// TIA Portal V19 export
DATA_BLOCK "A0302_PareggiatoreCoda"   // DB152
// stored: InstanceOfName A0302_PareggiatoreCoda_FB, InstanceOfType FB
"A0302_PareggiatoreCoda_FB"
   // VAR_INPUT
   //    AreaInterface : "AreaInterface";
   //    ZSI : "udt_ZoneSafetyInterface";
   //    DSI_Feed : "udt_DeviceSafetyInterface";
   //    DSI_Valve : "udt_DeviceSafetyInterface";
   //    DSI_OilValve : "udt_DeviceSafetyInterface";
   //    Drive : "TAx_DriveInterface";
   //    DataIn : Struct
   //       OP_MoveToPos : Bool;
   //       BattutaVrt : Struct
   //          OP : "OP_PB";
   //       END_STRUCT;
   //       PareggLong : Struct
   //          OP : "OP_PB";
   //          AnalSens : Int;
   //       END_STRUCT;
   //       Sens { ExternalWritable := 'False'} : Struct
   //          FTC_Ingombro_In : Bool;
   //          FTC_Ingombro_Out : Bool;
   //          PresenzaMat : Bool;
   //          FC_Aticoll_Spalla : Bool;
   //       END_STRUCT;
   //    END_STRUCT;
   //    CIn : Struct
   //       Manager : Struct
   //          EnableStopDoorOpeningReq { ExternalAccessible := 'False'; ExternalVisible := 'False'; ExternalWritable := 'False'} : Bool;
   //          EnableStopInPhase { ExternalAccessible := 'False'; ExternalVisible := 'False'; ExternalWritable := 'False'} : Bool;
   //          EnableStopProgrammed { ExternalAccessible := 'False'; ExternalVisible := 'False'; ExternalWritable := 'False'} : Bool;
   //          Control_ON { ExternalAccessible := 'False'; ExternalVisible := 'False'; ExternalWritable := 'False'} : Bool;
   //          MoveToPos { ExternalAccessible := 'False'; ExternalVisible := 'False'; ExternalWritable := 'False'} : Bool;
   //          Pos { ExternalAccessible := 'False'; ExternalVisible := 'False'; ExternalWritable := 'False'} : LReal;
   //          Speed : LReal;
   //          Bloccaggio { ExternalAccessible := 'False'; ExternalVisible := 'False'; ExternalWritable := 'False'} : Struct
   //             Rest : Bool;
   //             Work : Bool;
   //          END_STRUCT;
   //          BattutaVrt { ExternalAccessible := 'False'; ExternalVisible := 'False'; ExternalWritable := 'False'} : Struct
   //             Rest : Bool;
   //             Work : Bool;
   //          END_STRUCT;
   //          PareggLong { ExternalAccessible := 'False'; ExternalVisible := 'False'; ExternalWritable := 'False'} : Struct
   //             Rest : Bool;
   //             Work : Bool;
   //          END_STRUCT;
   //       END_STRUCT;
   //       SemiAut_Pb { ExternalWritable := 'False'} : Bool;
   //       Bordatrice : Struct
   //          Ax : "Positioning_EPOS_Machine_COut";
   //          Sts : Struct
   //             PosTargetEnable : Bool;
   //             PosTarget_Reached : Bool;
   //             In_W_Pos : Bool;
   //             AtRest : Bool;
   //          END_STRUCT;
   //          RegSpalla : Struct
   //             Infeed_ReqON : Bool;
   //          END_STRUCT;
   //       END_STRUCT;
   //       Rulliera { ExternalWritable := 'False'} : Struct
   //          Ax_1 : "SpeedMachine_COut";
   //          Ax_2 : "SpeedMachine_COut";
   //          Centratori : "ValveMachine_COut";
   //          Coda : Struct
   //             Sens : Struct
   //                FTC_Rall : Bool;
   //                FTC_Prox_Ing : Bool;
   //             END_STRUCT;
   //          END_STRUCT;
   //          Centro : Struct
   //             Sens : Struct
   //                FTC_Centrale : Bool;
   //             END_STRUCT;
   //          END_STRUCT;
   //       END_STRUCT;
   //       CarroPareggCoda : Struct
   //          Pareggia : Bool;
   //          OilInTargetPressure { ExternalWritable := 'False'} : Bool;
   //       END_STRUCT;
   //       CarroPareggTesta { ExternalWritable := 'False'} : Struct
   //          Sens : Struct
   //             FTC1_Rall : Bool;
   //             FTC2_Prox_Ls : Bool;
   //             PresenzaMat : Bool;
   //          END_STRUCT;
   //       END_STRUCT;
   //       CarriPareggiatori : Struct
   //          ZoneA0302Entry_Empty { ExternalWritable := 'False'} : Bool;
   //          ZoneA0302Exit_Empty { ExternalWritable := 'False'} : Bool;
   //          RequestNewPosition : Bool;
   //       END_STRUCT;
   //       Spalle : Struct
   //          Coda : Struct
   //             ActualPos : LReal;
   //          END_STRUCT;
   //          Testa : Struct
   //             ActualPos : LReal;
   //          END_STRUCT;
   //       END_STRUCT;
   //       Manipolatore : Struct
   //          Sollevatore : "ValveMachine_COut";
   //       END_STRUCT;
   //       Centratori : Struct
   //          Sollevamento : "ValveMachine_COut";
   //       END_STRUCT;
   //    END_STRUCT;
   //    Config : Struct
   //       Ax : "Positioning_DOL_Machine_Config";
   //       Bloccaggio : "ValveMachine_Config";
   //       BattutaVerticale : "ValveMachine_Config";
   //       PareggiatoreLong : "ValveMachine_Config";
   //       PosPareggiatore : Struct
   //          QuotaMin_Work : LReal;
   //          QuotaMax_Work : LReal;
   //       END_STRUCT;
   //       MinDistanzaConSpalla : LReal;
   //       DelayMissingCondition : Time;
   //    END_STRUCT;
   //    HWID : Struct
   //       Ax_TEL1 : HW_SUBMODULE;
   //       Enc_IO : HW_SUBMODULE;
   //    END_STRUCT;
   // END_VAR
   // VAR_OUTPUT
   //    MachineInterface : "MachineInterface";
   //    COut : Struct
   //       Ax : "Positioning_DOL_Machine_COut";
   //       Bloccaggio : "ValveMachine_COut";
   //       BattutaVerticale : "ValveMachine_COut";
   //       PareggiatoreLong : "ValveMachine_COut";
   //       Ax_InWPos : Bool;
   //       Anticipi : Struct
   //          Work : Struct
   //             BattutaVrt : Bool;
   //             PareggLong : Bool;
   //          END_STRUCT;
   //          Rest : Struct
   //             BattutaVrt : Bool;
   //             PareggLong : Bool;
   //          END_STRUCT;
   //       END_STRUCT;
   //    END_STRUCT;
   // END_VAR
   // VAR_IN_OUT
   //    Par : Struct
   //       Ax : "Positioning_DOL_Machine_Par";
   //       Ax_Pers : "Positioning_DOL_Machine_Pers_Data";
   //       Enc : "PosFbk_RTN";
   //       Ax_Aut : "A0301_Mach_Speed_Par";
   //       Bloccaggio_Sens : Struct
   //          "2191B1" : "Analogic_SensorManagement_Par";
   //          SogliaWork : Real;
   //       END_STRUCT;
   //       CarroPareggCoda : Struct
   //          Delay_StartMove : Time;
   //          Preset : LReal;
   //       END_STRUCT;
   //       Cremaliera : Struct
   //          Modulo : LReal;
   //          Passo : LReal;
   //       END_STRUCT;
   //    END_STRUCT;
   //    Par_Sens : Struct
   //       AI : "Analogic_SensorManagement_Par";
   //    END_STRUCT;
   //    Data_Sens : "Analogic_SensorManagement_Data";
   //    Par_MachSens : "A0301_Mach_Sens_Par";
   //    IEC_SP : Struct
   //       FTC_Input : Struct
   //          TON_PT : Time;
   //          TOF_PT : Time;
   //       END_STRUCT;
   //       FTC_Output : Struct
   //          TON_PT : Time;
   //          TOF_PT : Time;
   //       END_STRUCT;
   //       FTC_PresentMat : Struct
   //          TON_PT : Time;
   //          TOF_PT : Time;
   //       END_STRUCT;
   //       Check_2119B1 : Struct
   //          TON_PT : Time;
   //       END_STRUCT;
   //    END_STRUCT;
   // END_VAR
   // VAR
   //    Alarm : Struct
   //       Ax : "Positioning_DOL_Machine_Alr";
   //       Enc : "PosFbk_Encoder_Alr";
   //       Bloccaggio : "ValveAlr";
   //       BattutaVerticale : "ValveAlr";
   //       PareggiatoreLong : "ValveAlr";
   //       PareggLong_AnalSens_Issue : Bool;
   //       SensFC_Aticoll_Spalla : Bool;
   //       Bloccaggio_AnalSens_Issue : Bool;
   //    END_STRUCT;
   //    Warning : Struct
   //       Ax : "Positioning_DOL_Machine_Wng";
   //       Bloccaggio : "ValveMachine_Wng";
   //       BattutaVerticale : "ValveMachine_Wng";
   //       PareggiatoreLongitudinale : "ValveMachine_Wng";
   //       PosPareggiatoreLong : "Analogic_SensorManagement_Warning";
   //       MissingCnd : Struct
   //          OP_REST_BattutaVrt : Bool;
   //          OP_WORK_BattutaVrt : Bool;
   //          OP_REST_PareggLong : Bool;
   //          OP_WORK_PareggLong : Bool;
   //          OP_REST_Bloccaggio : Bool;
   //          OP_WORK_Bloccaggio : Bool;
   //       END_STRUCT;
   //       SW_Limit_AntiCollision : Bool;
   //    END_STRUCT;
   //    HMI : Struct
   //       AnalogSensor : "AnalogSens_HmiData";
   //       Ax : Struct
   //          PbPreset : Bool;
   //          B_Preset_UM2 : Bool;
   //          PresetValue : LReal;
   //       END_STRUCT;
   //    END_STRUCT;
   //    Sts : Struct
   //       ReadyForMove : Bool;
   //       OP_PCoda_CanMoveFreely : Bool;
   //       OP_Ax_CanMoveFreely : Bool;
   //       Op_MoveToPos_Cnd : Bool;
   //       BattutaVrt : Struct
   //          OP_Rest_Cnd : Bool;
   //          Op_Work_Cnd : Bool;
   //       END_STRUCT;
   //       PareggLong : Struct
   //          OP_Rest_Cnd : Bool;
   //          Op_Work_Cnd : Bool;
   //       END_STRUCT;
   //    END_STRUCT;
   //    Ctrl : Struct
   //       BattutaVrt : Struct
   //          OP_Rest_Man : Bool;
   //          OP_Work_Man : Bool;
   //          OP_Rest_Aut : Bool;
   //          OP_Work_Aut : Bool;
   //          OP_Rest : Bool;
   //          OP_Work : Bool;
   //       END_STRUCT;
   //       PareggLong : Struct
   //          CheckMesure : Bool;
   //          OP_Rest_Aut : Bool;
   //          OP_Work_Aut : Bool;
   //          OP_Rest_Man : Bool;
   //          OP_Work_Man : Bool;
   //          OP_Rest : Bool;
   //          OP_Work : Bool;
   //       END_STRUCT;
   //       Ax : Struct
   //          OP_MoveToPos_Man : Bool;
   //          OP_MoveToPos_Aut : Bool;
   //          OP_MoveToPos : Bool;
   //       END_STRUCT;
   //    END_STRUCT;
   //    AUX : Struct
   //       OP_MoveToPos : Bool;
   //       BattutaVrt : Struct
   //          OP_Rest : Bool;
   //          OP_Work : Bool;
   //       END_STRUCT;
   //       PareggLong : Struct
   //          OP_Rest : Bool;
   //          OP_Work : Bool;
   //       END_STRUCT;
   //    END_STRUCT;
   //    Ax { S7_SetPoint := 'True'} : "Positioning_DOL_Machine_FB";
   //    Enc : "PosFbk_SickAFM60";
   //    Enc_ITF : "PosFbk_ITF";
   //    Bloccaggio { S7_SetPoint := 'True'} : "ValveMachine_FB";
   //    BattutaVerticale { S7_SetPoint := 'True'} : "ValveMachine_FB";
   //    PareggiatoreLong { S7_SetPoint := 'True'} : "ValveMachine_FB";
   //    PosPareggLong { S7_SetPoint := 'True'} : "Analogic_SensorManagement";
   //    TON_PareggLong : Struct
   //       OP_REST_MissingCnd { S7_SetPoint := 'True'} : TON_TIME;
   //       OP_WORK_MissingCnd { S7_SetPoint := 'True'} : TON_TIME;
   //    END_STRUCT;
   //    TON_BattutaVrt : Struct
   //       OP_REST_MissingCnd { S7_SetPoint := 'True'} : TON_TIME;
   //       OP_WORK_MissingCnd { S7_SetPoint := 'True'} : TON_TIME;
   //    END_STRUCT;
   //    TON_Bloccaggio : Struct
   //       OP_REST_MissingCnd { S7_SetPoint := 'True'} : TON_TIME;
   //       OP_WORK_MissingCnd { S7_SetPoint := 'True'} : TON_TIME;
   //    END_STRUCT;
   //    IEC_FTC_Input : Struct
   //       TON_Delay : IEC_TIMER;
   //       TOF_Delay { S7_SetPoint := 'True'} : IEC_TIMER;
   //       FTC_On { S7_SetPoint := 'True'} : Bool;
   //    END_STRUCT;
   //    IEC_FTC_Output : Struct
   //       TON_Delay : IEC_TIMER;
   //       TOF_Delay { S7_SetPoint := 'True'} : IEC_TIMER;
   //       FTC_On { S7_SetPoint := 'True'} : Bool;
   //    END_STRUCT;
   //    IEC_FTC_PresentMat : Struct
   //       TON_Delay : IEC_TIMER;
   //       TOF_Delay { S7_SetPoint := 'True'} : IEC_TIMER;
   //       FTC_On { S7_SetPoint := 'True'} : Bool;
   //    END_STRUCT;
   //    IEC_DelayCheck_2119B1 : IEC_TIMER;
   //    Bloccaggio_AnalSens { S7_SetPoint := 'True'} : "AnalogThreshold";
   //    CarroCoda { ExternalAccessible := 'False'; ExternalVisible := 'False'; ExternalWritable := 'False'} : Struct
   //       RimanenzaPos : LReal;
   //       PassoReq : LReal;
   //       PosBattutePz : LReal;
   //       SemiBeamLen : LReal;
   //       NrPassiReq : LReal;
   //       Pos : LReal;
   //    END_STRUCT;
   //    TON_DistanzaOK : IEC_TIMER;
   //    TON_Anticipi : Struct
   //       Rest : Struct
   //          BattutaVrt { S7_SetPoint := 'True'} : IEC_TIMER;
   //          PareggLong : IEC_TIMER;
   //       END_STRUCT;
   //       Work : Struct
   //          PareggLong : IEC_TIMER;
   //          BattutaVrt { S7_SetPoint := 'True'} : IEC_TIMER;
   //       END_STRUCT;
   //    END_STRUCT;
   // END_VAR
BEGIN
END_DATA_BLOCK
